{attribute 'pack_mode' := '1'}
TYPE ST_SupervisorHeader :
	STRUCT
		{attribute 'hide'}
		Protocol_version : UINT := 4;
		{attribute 'hide'}
		Message_ID		 : UINT;
		{attribute 'hide'}
		Message_length	 : UDINT;
	END_STRUCT
END_TYPE

(* stored: Version 1.1.0.1, ProductVersion 3.1.4026.17
   DUT ST_SupervisorHeader: Id {77264308-66a8-4f31-8b94-b1e1812d84ee} *)
